INTERFACE I_XTS_Environment  EXTENDS __SYSTEM.IQueryInterface

{attribute 'monitoring':='call'}
PROPERTY HR : HRESULT
GET
END_GET
END_PROPERTY

METHOD Initialize : HRESULT
END_METHOD

{attribute 'monitoring':='call'}
PROPERTY TrackIsRing : BOOL
GET
END_GET
END_PROPERTY

{attribute 'monitoring':='call'}
PROPERTY TrackLength : LREAL
GET
END_GET
END_PROPERTY

METHOD Update : HRESULT
VAR_INPUT
END_VAR
END_METHOD

PROPERTY UtilityEnvirement : Tc3_XTS_Utility.i_TcIoXtsEnvironment
GET
END_GET
END_PROPERTY

END_INTERFACE

(* stored: Version 1.1.0.1, ProductVersion 3.1.4024.12
   Itf I_XTS_Environment: Id {0f1fffd3-3f82-4722-afce-252d61062d2b}
   Property HR: Id {bb8ae542-0b52-4660-9af1-4083d39a377b}
   Get Get: Id {32805057-8cbd-4c9e-b572-f4eba581e7aa}
   Method Initialize: Id {385eb571-6f87-4841-b5b8-894559f7775e}
   Property TrackIsRing: Id {4380e6d3-bcc4-4052-8fa7-b9b119deb435}
   Get Get: Id {eb78a3c6-cb92-4348-8347-9453f5ca9d4d}
   Property TrackLength: Id {db161dbe-a890-4d15-bf3c-281fdf1b0785}
   Get Get: Id {f606f0c2-4f64-4599-a50b-90e02365bb95}
   Method Update: Id {589f0e87-d0d0-4507-b1b4-133f8eede137}
   Property UtilityEnvirement: Id {02ce8ee7-e514-4db7-80ce-ba208a82fe2a}
   Get Get: Id {35794d32-aa7f-45ac-977f-73b302fb109e} *)
